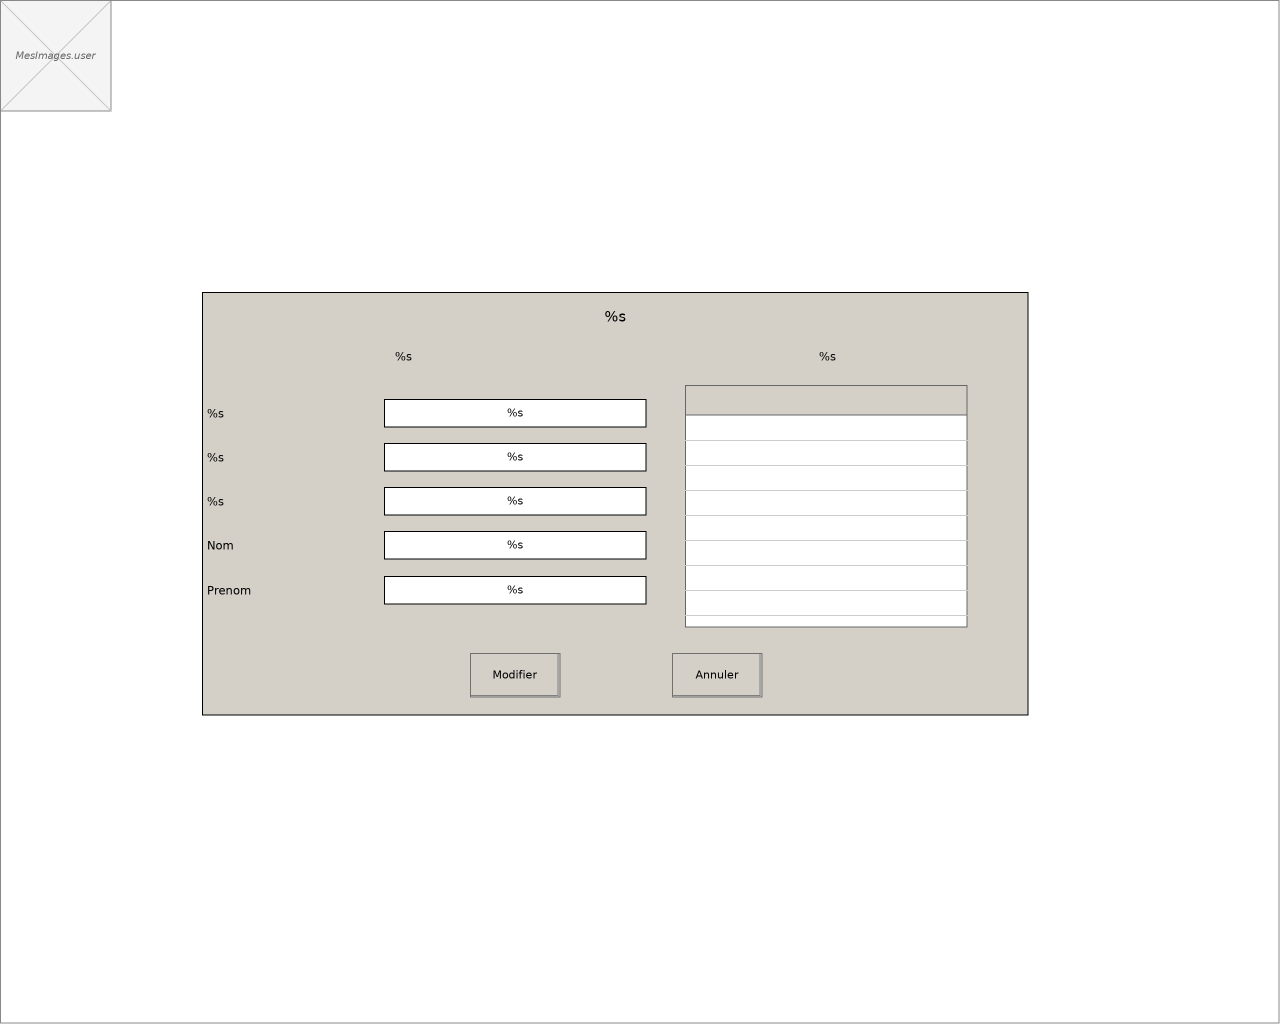
VISUALIZATION UTIL_MOD_USER  // 1280x1024
    Image (0,0 111x111), image: MesImages.user
    RoundedRectangle (202,292 826x423)
    Rectangle (206,302 819x29), "%s", text list: 'TextList_Util_Userlist', text index: 0
    Button (470,653 90x44), "Modifier", input disabled if: NOT PRG_USER.AUT_NOM_USER
        toggle PRG_USER.DD_mod_user2
        OnMouseClick: change screen: UTIL_USER
    Button (672,653 90x44), "Annuler"
        OnMouseClick: change screen: UTIL_USER
    Rectangle (384,399 262x28), "%s", text variable: PRG_USER.USER_TEMP.LOGIN
        OnMouseClick: write the text variable via InputWithLimits
    Rectangle (205,342 397x29), "%s", text list: 'TextList_Util_Userlist', text index: 2
    Rectangle (629,342 397x29), "%s", text list: 'TextList_Util_Userlist', text index: 3
    Table (685,385 282x242), data array: PRG_USER.TBL_GROUP
        p1137915858: PRG_USER.LIGNE_GROUP
        p3854506369: PRG_USER.TBL_GROUP[INDEX].NOM
        p1892666644: PRG_USER.TBL_GROUP[INDEX].PROGRAMMATION
        p338671338: PRG_USER.TBL_GROUP[INDEX].MAINTENANCE
        p2170511999: PRG_USER.TBL_GROUP[INDEX].SUPERVISEUR
        p3723444502: PRG_USER.TBL_GROUP[INDEX].PRODUCTION
        p1218418051: PRG_USER.TBL_GROUP[INDEX].CONF_MACHINE
        p746581629: PRG_USER.TBL_GROUP[INDEX].FONCTION_SA
        p3104783080: PRG_USER.TBL_GROUP[INDEX].CONF_TRF
        p2501879983: PRG_USER.TBL_GROUP[INDEX].MODIF_ENLIGNE
        p7306298: PRG_USER.TBL_GROUP[INDEX].ARCHIVE_EV
        p1933151965: PRG_USER.TBL_GROUP[INDEX].DECONSIGNATION
        p2232123230: Nom du groupe
        p511219082: Pro. Ed
        p1755163831: Maint.
        p4092479075: Superv.
        p2237128397: Prod.
        p505689113: Conf.
        p1757482276: FoncSA.
    Rectangle (204,399 173x29), "%s", text list: 'TextList_Users_Menu', text index: 5
    Rectangle (204,443 173x29), "%s", text list: 'TextList_Users_Menu', text index: 6
    Rectangle (204,487 173x29), "%s", text list: 'TextList_Users_Menu', text index: 21
    Rectangle (204,531 173x29), "Nom"
    Rectangle (204,576 173x29), "Prenom"
    Rectangle (384,443 262x28), "%s", text variable: PRG_USER.USER_TEMP.PASS
        OnMouseClick: write the text variable via InputWithLimits, password
    Rectangle (384,487 262x28), "%s", text variable: PRG_USER.PASS_CONF
        OnMouseClick: write the text variable via InputWithLimits, password
    Rectangle (384,531 262x28), "%s", text variable: PRG_USER.USER_TEMP.NOM
        OnMouseClick: write the text variable via InputWithLimits
    Rectangle (384,576 262x28), "%s", text variable: PRG_USER.USER_TEMP.PRENOM
        OnMouseClick: write the text variable via InputWithLimits
END_VISUALIZATION

(* stored: Version 1.1.0.1, ProductVersion 3.1.4024.10
   Visu UTIL_MOD_USER: Id {3fd53a47-9f22-466e-b85b-a87849f1f47d} *)
